FUNCTION TryConvert_DINT_TO_BOOL : BOOL
VAR_INPUT
	in : DINT;
	out : REFERENCE TO BOOL;
END_VAR

out := DINT_TO_BOOL(in);
TryConvert_DINT_TO_BOOL := TRUE;

END_FUNCTION

(* stored: Version 1.1.0.1, ProductVersion 3.1.4024.12
   POU TryConvert_DINT_TO_BOOL: Id {cd260842-bd8f-43d0-88ae-2285a19f8f11}, SpecialFunc None *)
